PROGRAM Systemparameter
VAR
END_VAR

// Lesen
	// Objektzustände
	GVL.Robot_State 		:= Anlage.UR5.P_State;
	GVL.Greifer_State 		:= Anlage.Gripper.P_State;
	GVL.Sensor_State 		:= 1;

// Zuweisen
	// Eigenschaften	
	Anlage.HEX_E.P_LimitValue 		:= GVL.eKraftLimitValue;
	Anlage.HEX_E.P_ErreichtValue 	:= GVL.eKraftErreichtValue;

END_PROGRAM

(* stored: Version 1.1.0.1
   POU Systemparameter: Id {2b7e68ef-f113-4809-903c-9cd92fcb2e25}, SpecialFunc None *)
